(* IEC 61131-3 sources: smart-traffic-light/tests, 11 files *)

(* ---- test_data_types.st ---- *)
(* Tests for traffic light data types *)

TEST 'TrafficState enum values are distinct'
  VAR
    s1 : TrafficState;
    s2 : TrafficState;
    s3 : TrafficState;
  END_VAR

  s1 := TrafficState.RED;
  s2 := TrafficState.YELLOW;
  s3 := TrafficState.GREEN;

  ASSERT_NEQ(s1, s2, 'RED and YELLOW must differ');
  ASSERT_NEQ(s2, s3, 'YELLOW and GREEN must differ');
  ASSERT_NEQ(s1, s3, 'RED and GREEN must differ');
END_TEST

TEST 'PedestrianState enum values are distinct'
  VAR
    p1 : PedestrianState;
    p2 : PedestrianState;
    p3 : PedestrianState;
  END_VAR

  p1 := PedestrianState.WALK;
  p2 := PedestrianState.DONT_WALK;
  p3 := PedestrianState.FLASHING;

  ASSERT_NEQ(p1, p2, 'WALK and DONT_WALK must differ');
  ASSERT_NEQ(p2, p3, 'DONT_WALK and FLASHING must differ');
END_TEST

TEST 'PhaseTiming struct default values'
  VAR timing : PhaseTiming; END_VAR

  ASSERT_EQ(timing.greenDuration, T#30s, 'Default green should be 30s');
  ASSERT_EQ(timing.yellowDuration, T#5s, 'Default yellow should be 5s');
  ASSERT_EQ(timing.redDuration, T#35s, 'Default red should be 35s');
END_TEST

TEST 'PhaseTiming struct custom values'
  VAR timing : PhaseTiming; END_VAR

  timing.greenDuration := T#20s;
  timing.yellowDuration := T#3s;
  timing.redDuration := T#25s;

  ASSERT_EQ(timing.greenDuration, T#20s);
  ASSERT_EQ(timing.yellowDuration, T#3s);
  ASSERT_EQ(timing.redDuration, T#25s);
END_TEST

TEST 'LogEntry struct initialization'
  VAR entry : LogEntry; END_VAR

  entry.previousState := TrafficState.RED;
  entry.newState := TrafficState.GREEN;
  entry.timestamp := T#1500ms;

  ASSERT_EQ(entry.previousState, TrafficState.RED);
  ASSERT_EQ(entry.newState, TrafficState.GREEN);
  ASSERT_EQ(entry.timestamp, T#1500ms);
END_TEST

(* ---- test_interface.st ---- *)
(* Tests for IControllable interface implementation *)

TEST 'TrafficLight implements Enable method'
  VAR light : TrafficLight; END_VAR

  light.active := FALSE;
  light();
  ASSERT_FALSE(light.IsEnabled(), 'Should be disabled');

  light.Enable();
  ASSERT_TRUE(light.IsEnabled(), 'Should be enabled after Enable()');
END_TEST

TEST 'TrafficLight implements Disable method'
  VAR light : TrafficLight; END_VAR

  light();
  ASSERT_TRUE(light.IsEnabled(), 'Enabled by default');

  light.Disable();
  ASSERT_FALSE(light.IsEnabled(), 'Disabled after Disable()');
END_TEST

TEST 'TrafficLight GetStatus returns correct codes'
  VAR
    light  : TrafficLight;
    timing : PhaseTiming;
  END_VAR

  timing.redDuration := T#100ms;
  timing.greenDuration := T#100ms;
  timing.yellowDuration := T#50ms;
  light.timing := timing;

  (* Disabled state *)
  light.active := FALSE;
  light();
  ASSERT_EQ(light.GetStatus(), 0, 'Disabled = 0');

  (* RED state *)
  light.active := TRUE;
  light();
  ASSERT_EQ(light.GetStatus(), 1, 'RED = 1');

  (* Night mode *)
  light.nightMode := TRUE;
  light();
  ASSERT_EQ(light.GetStatus(), 4, 'Night mode = 4');
END_TEST

(* ---- test_night_mode.st ---- *)
(* Tests for TrafficLight night mode feature *)

TEST 'Night mode turns off red and green lights'
  VAR light : TrafficLight; END_VAR

  light.nightMode := TRUE;
  light();

  ASSERT_FALSE(light.redLight, 'Red should be off in night mode');
  ASSERT_FALSE(light.greenLight, 'Green should be off in night mode');
END_TEST

TEST 'Night mode sets state to YELLOW'
  VAR light : TrafficLight; END_VAR

  light.nightMode := TRUE;
  light();

  ASSERT_EQ(light.currentState, TrafficState.YELLOW, 'State should be YELLOW in night mode');
END_TEST

TEST 'Night mode flashes yellow'
  VAR light : TrafficLight; END_VAR

  light.nightMode := TRUE;
  light();

  (* After first flash period *)
  ADVANCE_TIME(T#500ms);
  light();

  (* Yellow should have toggled *)
  ASSERT_EQ(light.currentState, TrafficState.YELLOW, 'Still in YELLOW state');
END_TEST

TEST 'Exiting night mode resumes normal operation'
  VAR
    light  : TrafficLight;
    timing : PhaseTiming;
  END_VAR

  timing.redDuration := T#100ms;
  timing.greenDuration := T#100ms;
  timing.yellowDuration := T#50ms;
  light.timing := timing;

  (* Enter night mode *)
  light.nightMode := TRUE;
  light();
  ADVANCE_TIME(T#200ms);
  light();

  (* Exit night mode *)
  light.nightMode := FALSE;
  light();

  (* Should resume normal cycling from YELLOW state *)
  ASSERT_FALSE(light.nightMode, 'Night mode should be off');
END_TEST

TEST 'IsNightMode method returns correct state'
  VAR light : TrafficLight; END_VAR

  light();
  ASSERT_FALSE(light.IsNightMode(), 'Not in night mode initially');

  light.nightMode := TRUE;
  light();
  ASSERT_TRUE(light.IsNightMode(), 'Should report night mode');
END_TEST

(* ---- test_pedestrian_light.st ---- *)
(* Tests for the PedestrianLight function block *)

TEST 'PedestrianLight starts in DONT_WALK'
  VAR ped : PedestrianLight; END_VAR

  ped();
  ASSERT_EQ(ped.pedestrianState, PedestrianState.DONT_WALK, 'Should start DONT_WALK');
  ASSERT_TRUE(ped.dontWalkLight, 'Dont walk light should be on');
  ASSERT_FALSE(ped.walkLight, 'Walk light should be off');
END_TEST

TEST 'PedestrianLight walks when traffic is RED and requested'
  VAR
    ped : PedestrianLight;
    timing : PhaseTiming;
  END_VAR

  timing.redDuration := T#200ms;
  timing.greenDuration := T#100ms;
  timing.yellowDuration := T#50ms;
  ped.timing := timing;
  ped.walkDuration := T#80ms;

  (* Start in RED *)
  ped();
  ASSERT_EQ(ped.currentState, TrafficState.RED, 'Should be RED');

  (* Request walk *)
  ped.walkRequest := TRUE;
  ped();

  ASSERT_EQ(ped.pedestrianState, PedestrianState.WALK, 'Should be WALK after request during RED');
  ASSERT_TRUE(ped.walkLight, 'Walk light should be on');
END_TEST

TEST 'PedestrianLight transitions WALK to FLASHING after duration'
  VAR
    ped : PedestrianLight;
    timing : PhaseTiming;
  END_VAR

  timing.redDuration := T#500ms;
  timing.greenDuration := T#100ms;
  timing.yellowDuration := T#50ms;
  ped.timing := timing;
  ped.walkDuration := T#80ms;

  ped.walkRequest := TRUE;
  ped();
  ASSERT_EQ(ped.pedestrianState, PedestrianState.WALK, 'Should be WALK');

  (* Advance past walk duration *)
  ADVANCE_TIME(T#40ms);
  ped();
  ADVANCE_TIME(T#40ms);
  ped();

  ASSERT_EQ(ped.pedestrianState, PedestrianState.FLASHING, 'Should be FLASHING after walk duration');
END_TEST

TEST 'PedestrianLight IsWalking method'
  VAR
    ped : PedestrianLight;
    timing : PhaseTiming;
  END_VAR

  timing.redDuration := T#200ms;
  ped.timing := timing;

  ped();
  ASSERT_FALSE(ped.IsWalking(), 'Not walking initially');

  ped.walkRequest := TRUE;
  ped();
  ASSERT_TRUE(ped.IsWalking(), 'Walking after request during RED');
END_TEST

TEST 'PedestrianLight resets when traffic goes GREEN'
  VAR
    ped : PedestrianLight;
    timing : PhaseTiming;
  END_VAR

  timing.redDuration := T#100ms;
  timing.greenDuration := T#100ms;
  timing.yellowDuration := T#50ms;
  ped.timing := timing;

  (* Walk during RED *)
  ped.walkRequest := TRUE;
  ped();
  ASSERT_EQ(ped.pedestrianState, PedestrianState.WALK);

  (* Advance to GREEN *)
  ADVANCE_TIME(T#50ms);
  ped();
  ADVANCE_TIME(T#50ms);
  ped();

  ASSERT_EQ(ped.currentState, TrafficState.GREEN, 'Traffic should be GREEN');
  ASSERT_EQ(ped.pedestrianState, PedestrianState.DONT_WALK, 'Ped should be DONT_WALK');
  ASSERT_FALSE(ped.walkRequest, 'Walk request should be cleared');
END_TEST

(* ---- test_pedestrian_timeout_fix.st ---- *)
(* Tests for pedestrian timeout fix — verifies timer reset on state change *)

TEST 'Walk timer resets when traffic leaves RED'
  VAR
    ped : PedestrianLight;
    timing : PhaseTiming;
  END_VAR

  timing.redDuration := T#500ms;
  timing.greenDuration := T#100ms;
  timing.yellowDuration := T#50ms;
  ped.timing := timing;
  ped.walkDuration := T#200ms;

  (* Start walking during RED *)
  ped.walkRequest := TRUE;
  ped();
  ASSERT_EQ(ped.pedestrianState, PedestrianState.WALK, 'Walking during RED');

  (* Advance partially through walk duration *)
  ADVANCE_TIME(T#50ms);
  ped();

  (* Force traffic to GREEN by advancing past red duration *)
  ADVANCE_TIME(T#450ms);
  ped();
  ASSERT_EQ(ped.currentState, TrafficState.GREEN, 'Traffic now GREEN');
  ASSERT_EQ(ped.pedestrianState, PedestrianState.DONT_WALK, 'Walk cancelled');

  (* Go through GREEN + YELLOW back to RED *)
  ADVANCE_TIME(T#50ms);
  ped();
  ADVANCE_TIME(T#50ms);
  ped();
  ADVANCE_TIME(T#25ms);
  ped();
  ADVANCE_TIME(T#25ms);
  ped();

  (* Should be back in RED now *)
  ASSERT_EQ(ped.currentState, TrafficState.RED, 'Back to RED');

  (* Request walk again during new RED phase *)
  ped.walkRequest := TRUE;
  ped();
  ASSERT_EQ(ped.pedestrianState, PedestrianState.WALK, 'Can walk again');

  (* Walk timer should start fresh, not carry over old elapsed time.
     Only 100ms elapsed out of 200ms duration — should still be walking. *)
  ADVANCE_TIME(T#100ms);
  ped();
  ASSERT_EQ(ped.pedestrianState, PedestrianState.WALK,
    'Still walking — timer was properly reset');
END_TEST

TEST 'Flash timer resets when traffic leaves RED'
  VAR
    ped : PedestrianLight;
    timing : PhaseTiming;
  END_VAR

  timing.redDuration := T#500ms;
  timing.greenDuration := T#100ms;
  timing.yellowDuration := T#50ms;
  ped.timing := timing;
  ped.walkDuration := T#50ms;

  (* Walk and transition to flashing *)
  ped.walkRequest := TRUE;
  ped();
  ADVANCE_TIME(T#25ms);
  ped();
  ADVANCE_TIME(T#25ms);
  ped();
  ASSERT_EQ(ped.pedestrianState, PedestrianState.FLASHING, 'Should be flashing');

  (* Simulate early exit — flash count and timer should reset cleanly *)
  ped.walkRequest := FALSE;
  ped();

  (* Re-request walk *)
  ped.walkRequest := TRUE;
  ped();
  ASSERT_EQ(ped.pedestrianState, PedestrianState.WALK, 'Fresh walk cycle');
END_TEST

(* ---- test_safety_validation.st ---- *)
(* Safety validation tests — ensure timing parameters meet minimum requirements *)

TEST 'Default yellow duration meets minimum safety threshold'
  VAR timing : PhaseTiming; END_VAR

  (* Federal Highway Administration recommends minimum 3s yellow for
     intersections with speed limits up to 25 mph. This test enforces
     that the default yellow duration is at least 3 seconds. *)
  ASSERT_TRUE(timing.yellowDuration >= T#3s,
    'Yellow duration must be at least 3s for safety');
END_TEST

TEST 'Default green duration is reasonable'
  VAR timing : PhaseTiming; END_VAR

  ASSERT_TRUE(timing.greenDuration >= T#10s,
    'Green duration should be at least 10s');
  ASSERT_TRUE(timing.greenDuration <= T#120s,
    'Green duration should not exceed 120s');
END_TEST

TEST 'Default red duration is reasonable'
  VAR timing : PhaseTiming; END_VAR

  ASSERT_TRUE(timing.redDuration >= T#10s,
    'Red duration should be at least 10s');
END_TEST

TEST 'Total cycle time is within bounds'
  VAR timing : PhaseTiming; END_VAR

  ASSERT_TRUE(
    timing.greenDuration + timing.yellowDuration + timing.redDuration >= T#30s,
    'Total cycle should be at least 30s');
  ASSERT_TRUE(
    timing.greenDuration + timing.yellowDuration + timing.redDuration <= T#300s,
    'Total cycle should not exceed 300s');
END_TEST

(* ---- test_timing_utils.st ---- *)
(* Tests for TimingUtils functions *)

TEST 'CalculateCycleTime sums all durations'
  VAR
    phases : ARRAY[1..3] OF TIME := [T#30s, T#5s, T#35s];
    total  : TIME;
  END_VAR

  total := CalculateCycleTime(phases);
  ASSERT_EQ(total, T#70s, 'Total cycle should be 70s');
END_TEST

TEST 'CalculateCycleTime with single phase'
  VAR
    phases : ARRAY[1..1] OF TIME := [T#45s];
    total  : TIME;
  END_VAR

  total := CalculateCycleTime(phases);
  ASSERT_EQ(total, T#45s, 'Single phase cycle');
END_TEST

TEST 'FindLongestPhase returns maximum duration'
  VAR
    phases  : ARRAY[1..3] OF TIME := [T#30s, T#5s, T#35s];
    longest : TIME;
  END_VAR

  longest := FindLongestPhase(phases);
  ASSERT_EQ(longest, T#35s, 'Longest should be 35s');
END_TEST

TEST 'ValidateMinDurations passes when all above threshold'
  VAR
    phases : ARRAY[1..3] OF TIME := [T#30s, T#5s, T#35s];
    valid  : BOOL;
  END_VAR

  valid := ValidateMinDurations(phases, T#3s);
  ASSERT_TRUE(valid, 'All durations above 3s');
END_TEST

TEST 'ValidateMinDurations fails when one below threshold'
  VAR
    phases : ARRAY[1..3] OF TIME := [T#30s, T#2s, T#35s];
    valid  : BOOL;
  END_VAR

  valid := ValidateMinDurations(phases, T#3s);
  ASSERT_FALSE(valid, 'One duration below 3s');
END_TEST

TEST 'ScaleDuration doubles at 200 percent'
  VAR result : TIME; END_VAR

  result := ScaleDuration(T#10s, 200);
  ASSERT_EQ(result, T#20s, 'Should be doubled');
END_TEST

TEST 'ScaleDuration halves at 50 percent'
  VAR result : TIME; END_VAR

  result := ScaleDuration(T#10s, 50);
  ASSERT_EQ(result, T#5s, 'Should be halved');
END_TEST

(* ---- test_traffic_light.st ---- *)
(* Tests for the TrafficLight function block *)

TEST 'TrafficLight starts in RED state'
  VAR light : TrafficLight; END_VAR

  light();
  ASSERT_EQ(light.currentState, TrafficState.RED, 'Should start in RED');
  ASSERT_TRUE(light.redLight, 'Red light should be on');
  ASSERT_FALSE(light.greenLight, 'Green light should be off');
  ASSERT_FALSE(light.yellowLight, 'Yellow light should be off');
END_TEST

TEST 'TrafficLight transitions RED to GREEN after red duration'
  VAR
    light : TrafficLight;
    timing : PhaseTiming;
  END_VAR

  timing.redDuration := T#100ms;
  timing.greenDuration := T#100ms;
  timing.yellowDuration := T#50ms;
  light.timing := timing;

  (* Run through the red phase *)
  light();
  ADVANCE_TIME(T#50ms);
  light();
  ASSERT_EQ(light.currentState, TrafficState.RED, 'Still RED at 50ms');

  ADVANCE_TIME(T#50ms);
  light();
  ASSERT_EQ(light.currentState, TrafficState.GREEN, 'Should be GREEN after 100ms');
  ASSERT_TRUE(light.greenLight);
  ASSERT_FALSE(light.redLight);
END_TEST

TEST 'TrafficLight full cycle RED -> GREEN -> YELLOW -> RED'
  VAR
    light : TrafficLight;
    timing : PhaseTiming;
  END_VAR

  timing.redDuration := T#100ms;
  timing.greenDuration := T#80ms;
  timing.yellowDuration := T#40ms;
  light.timing := timing;

  (* Start in RED *)
  light();
  ASSERT_EQ(light.currentState, TrafficState.RED);

  (* Advance past red duration -> GREEN *)
  ADVANCE_TIME(T#50ms);
  light();
  ADVANCE_TIME(T#50ms);
  light();
  ASSERT_EQ(light.currentState, TrafficState.GREEN, 'After red duration -> GREEN');

  (* Advance past green duration -> YELLOW *)
  ADVANCE_TIME(T#40ms);
  light();
  ADVANCE_TIME(T#40ms);
  light();
  ASSERT_EQ(light.currentState, TrafficState.YELLOW, 'After green duration -> YELLOW');

  (* Advance past yellow duration -> RED *)
  ADVANCE_TIME(T#20ms);
  light();
  ADVANCE_TIME(T#20ms);
  light();
  ASSERT_EQ(light.currentState, TrafficState.RED, 'After yellow duration -> back to RED');
END_TEST

TEST 'TrafficLight disabled does not advance'
  VAR
    light : TrafficLight;
    timing : PhaseTiming;
  END_VAR

  timing.redDuration := T#100ms;
  light.timing := timing;
  light.active := FALSE;

  light();
  ADVANCE_TIME(T#200ms);
  light();

  ASSERT_EQ(light.currentState, TrafficState.RED, 'Disabled light should stay in RED');
END_TEST

TEST 'TrafficLight methods report correct state'
  VAR light : TrafficLight; END_VAR

  light();
  ASSERT_TRUE(light.IsRed(), 'IsRed should be TRUE initially');
  ASSERT_FALSE(light.IsGreen(), 'IsGreen should be FALSE initially');
  ASSERT_EQ(light.GetState(), TrafficState.RED, 'GetState should return RED');
END_TEST

(* ---- test_traffic_logger.st ---- *)
(* Tests for the TrafficLogger function block *)

TEST 'TrafficLogger starts empty'
  VAR logger : TrafficLogger; END_VAR

  ASSERT_EQ(logger.entryCount, 0, 'Should start empty');
  ASSERT_FALSE(logger.isFull, 'Should not be full');
END_TEST

TEST 'TrafficLogger requires initialization'
  VAR
    logger : TrafficLogger;
    ok     : BOOL;
  END_VAR

  ok := logger.LogTransition(TrafficState.RED, TrafficState.GREEN, T#1s);
  ASSERT_FALSE(ok, 'Should fail without init');

  ok := logger.Initialize();
  ASSERT_TRUE(ok, 'Initialize should succeed');

  ok := logger.LogTransition(TrafficState.RED, TrafficState.GREEN, T#1s);
  ASSERT_TRUE(ok, 'Should succeed after init');
  ASSERT_EQ(logger.entryCount, 1);

  logger.Cleanup();
END_TEST

TEST 'TrafficLogger counts entries'
  VAR
    logger : TrafficLogger;
    ok     : BOOL;
  END_VAR

  logger.Initialize();

  logger.LogTransition(TrafficState.RED, TrafficState.GREEN, T#1s);
  logger.LogTransition(TrafficState.GREEN, TrafficState.YELLOW, T#31s);
  logger.LogTransition(TrafficState.YELLOW, TrafficState.RED, T#36s);

  ASSERT_EQ(logger.entryCount, 3, 'Should have 3 entries');
  ASSERT_EQ(logger.GetTotalTransitions(), 3, 'Total should be 3');
  ASSERT_FALSE(logger.isFull, 'Should not be full with 3/20 entries');

  logger.Cleanup();
END_TEST

TEST 'TrafficLogger wraps around when full'
  VAR
    logger : TrafficLogger;
    i      : INT;
  END_VAR

  logger.bufferSize := 3;
  logger.Initialize();

  (* Fill the buffer *)
  logger.LogTransition(TrafficState.RED, TrafficState.GREEN, T#1s);
  logger.LogTransition(TrafficState.GREEN, TrafficState.YELLOW, T#31s);
  logger.LogTransition(TrafficState.YELLOW, TrafficState.RED, T#36s);

  ASSERT_TRUE(logger.isFull, 'Should be full at capacity');
  ASSERT_EQ(logger.entryCount, 3, 'Entry count capped at buffer size');

  (* Overwrite oldest entry *)
  logger.LogTransition(TrafficState.RED, TrafficState.GREEN, T#71s);
  ASSERT_EQ(logger.entryCount, 3, 'Still capped at 3');
  ASSERT_EQ(logger.GetTotalTransitions(), 4, 'Total includes overwritten');

  logger.Cleanup();
END_TEST

TEST 'TrafficLogger cleanup resets state'
  VAR logger : TrafficLogger; END_VAR

  logger.Initialize();
  logger.LogTransition(TrafficState.RED, TrafficState.GREEN, T#1s);
  logger.Cleanup();

  ASSERT_EQ(logger.entryCount, 0, 'Count reset after cleanup');
  ASSERT_FALSE(logger.isFull, 'Not full after cleanup');
END_TEST

(* ---- test_turn_signal.st ---- *)
(* Tests for the TurnSignalLight function block *)

TEST 'TurnSignalLight starts with arrow off'
  VAR ts : TurnSignalLight; END_VAR

  ts();
  ASSERT_FALSE(ts.turnArrowOn, 'Arrow should be off initially');
  ASSERT_EQ(ts.turnDirection, 0, 'No direction set');
END_TEST

TEST 'TurnSignalLight SetLeftTurn sets direction'
  VAR ts : TurnSignalLight; END_VAR

  ts.SetLeftTurn();
  ASSERT_EQ(ts.turnDirection, 1, 'Should be left turn');
END_TEST

TEST 'TurnSignalLight SetRightTurn sets direction'
  VAR ts : TurnSignalLight; END_VAR

  ts.SetRightTurn();
  ASSERT_EQ(ts.turnDirection, 2, 'Should be right turn');
END_TEST

TEST 'TurnSignalLight activates on RED to GREEN transition'
  VAR
    ts     : TurnSignalLight;
    timing : PhaseTiming;
  END_VAR

  timing.redDuration := T#100ms;
  timing.greenDuration := T#200ms;
  timing.yellowDuration := T#50ms;
  ts.timing := timing;
  ts.turnDuration := T#80ms;
  ts.SetLeftTurn();

  (* Start in RED *)
  ts();
  ASSERT_EQ(ts.currentState, TrafficState.RED, 'Start in RED');
  ASSERT_FALSE(ts.turnArrowOn, 'Arrow off during RED');

  (* Transition to GREEN *)
  ADVANCE_TIME(T#50ms);
  ts();
  ADVANCE_TIME(T#50ms);
  ts();
  ASSERT_EQ(ts.currentState, TrafficState.GREEN, 'Now GREEN');
  ASSERT_TRUE(ts.turnArrowOn, 'Arrow on during GREEN after RED');
END_TEST

TEST 'TurnSignalLight arrow turns off after duration'
  VAR
    ts     : TurnSignalLight;
    timing : PhaseTiming;
  END_VAR

  timing.redDuration := T#100ms;
  timing.greenDuration := T#300ms;
  timing.yellowDuration := T#50ms;
  ts.timing := timing;
  ts.turnDuration := T#80ms;
  ts.SetLeftTurn();

  (* Get to GREEN *)
  ts();
  ADVANCE_TIME(T#50ms);
  ts();
  ADVANCE_TIME(T#50ms);
  ts();
  ASSERT_TRUE(ts.turnArrowOn, 'Arrow should be on');

  (* Wait for turn duration to expire *)
  ADVANCE_TIME(T#40ms);
  ts();
  ADVANCE_TIME(T#40ms);
  ts();
  ASSERT_FALSE(ts.turnArrowOn, 'Arrow should be off after duration');
END_TEST

TEST 'TurnSignalLight IsTurnActive method'
  VAR ts : TurnSignalLight; END_VAR

  ts();
  ASSERT_FALSE(ts.IsTurnActive(), 'Not active initially');
END_TEST

(* ---- test_vehicle_detector.st ---- *)
(* Tests for the VehicleDetector function block *)

TEST 'VehicleDetector starts with zero count'
  VAR det : VehicleDetector; END_VAR

  det();
  ASSERT_EQ(det.vehicleCount, 0, 'Count should start at 0');
  ASSERT_FALSE(det.isOccupied, 'Not occupied initially');
END_TEST

TEST 'VehicleDetector counts on rising edge'
  VAR det : VehicleDetector; END_VAR

  det();

  (* First vehicle *)
  det.sensorInput := TRUE;
  det();
  ASSERT_EQ(det.vehicleCount, 1, 'One vehicle detected');
  ASSERT_TRUE(det.isOccupied, 'Should be occupied');

  (* Sensor still active — no new count *)
  det();
  ASSERT_EQ(det.vehicleCount, 1, 'Still one vehicle');

  (* Vehicle leaves *)
  det.sensorInput := FALSE;
  det();
  ASSERT_FALSE(det.isOccupied, 'No longer occupied');

  (* Second vehicle *)
  det.sensorInput := TRUE;
  det();
  ASSERT_EQ(det.vehicleCount, 2, 'Two vehicles total');
END_TEST

TEST 'VehicleDetector Initialize and Cleanup'
  VAR
    det : VehicleDetector;
    ok  : BOOL;
  END_VAR

  ok := det.Initialize();
  ASSERT_TRUE(ok, 'First initialize should succeed');

  ok := det.Initialize();
  ASSERT_FALSE(ok, 'Second initialize should fail (already init)');

  ok := det.Cleanup();
  ASSERT_TRUE(ok, 'Cleanup should succeed');

  ok := det.Cleanup();
  ASSERT_FALSE(ok, 'Second cleanup should fail (already cleaned)');
END_TEST

TEST 'VehicleDetector Reset clears count'
  VAR det : VehicleDetector; END_VAR

  det.sensorInput := TRUE;
  det();
  det.sensorInput := FALSE;
  det();
  det.sensorInput := TRUE;
  det();
  ASSERT_EQ(det.vehicleCount, 2, 'Should have 2 vehicles');

  det.Reset();
  ASSERT_EQ(det.vehicleCount, 0, 'Should be reset to 0');
  ASSERT_FALSE(det.isOccupied, 'Not occupied after reset');
END_TEST

TEST 'VehicleDetector GetDetectionCount method'
  VAR det : VehicleDetector; END_VAR

  det.sensorInput := TRUE;
  det();
  ASSERT_EQ(det.GetDetectionCount(), 1, 'Method should return count');
END_TEST
